PROGRAM MAIN
VAR
END_VAR

END_PROGRAM

(* stored: Version 1.1.0.1, ProductVersion 3.1.4024.12
   POU MAIN: Id {58a55f22-a46e-0bc8-2353-eea328b832b2}, SpecialFunc None *)
